{attribute 'hide_all_locals' := ''}
{attribute 'FBVisuCreatorPrefix' := 'RET_VISU_'}
FUNCTION_BLOCK Rauschen
VAR_INPUT
	{attribute 'FBVisuCreatorFormatString' := '%1.3f'}
	fVerstaerkung: REAL;
END_VAR
VAR_OUTPUT
	{attribute 'FBVisuCreatorFormatString' := '%1.3f'}
	fY: REAL;
END_VAR
VAR
	{attribute 'hide'}
	fSumme: REAL;
	{attribute 'hide'}
	nI: INT := 0;
END_VAR
VAR CONSTANT
	{attribute 'hide'}
